(* Logix 5000 project; controller LeakTestAuto vendor 1 type 14 code 226 rev 37.11; software revision 37.01; part 8 of 12 *)
(* tags used below, declared in another part *)
   AOI_Conveyor_Seq : AOI_Sequencer_x64;
   AOI_CTS2 : AOI_CTS_INSTRUMENT;
   AOI_CTS2_Comms : AOI_CommStatus;
   AOI_CTS2_Seq : AOI_Sequencer_x64;
   AOI_Robot_Comms : AOI_CommStatus;
   AOI_RobotPos : AOI_RobotPositions;
   AOI_SeqSteps : AOI_StandardSeqSteps;
   Conveyor : udt_OutputStructure;
   Conveyor_Seq : udt_SequenceStructure_X64;
   ConveyorCleatSensorFault : BOOL;
   CTS2_BarcodeWrite : STRING80;
   CTS2_BasicResult : MESSAGE;
   CTS2_DataRead : STRING80;
   CTS2_DetailResult : MESSAGE;
   CTS2_Inputs : udt_CTS_INPUTS_FROM;
   CTS2_LastResultEval : STRING16;
   CTS2_LastTestUID : DINT;
   CTS2_NextTestUID : DINT;
   CTS2_NumTestsInSeq : SINT;
   CTS2_Outputs : udt_CTS_OUTPUTS_TO;
   CTS2_ReadMsg : MESSAGE;
   CTS2_Ready : DINT;
   CTS2_Result : udt_CTS_RESULT;
   CTS2_ResultHistoryLeak : udt_CTS_RESULT[10];
   CTS2_ResultHistoryVol : udt_CTS_RESULT[10];
   CTS2_Seq : udt_SequenceStructure_X64;
   CTS2_SeqUID : DINT;
   CTS2_UIDMsg : MESSAGE;
   CTS2_WriteMsg : MESSAGE;
   CTS_NoResult : udt_CTS_RESULT;
   CTS_ResultDump : udt_CTS_RESULT;
   CurrentDUTData : udt_DUTHistory[2];
   FFLU_CTS2Leak : CONTROL;
   FFLU_CTS2Vol : CONTROL;
   LeakTester2 : udt_OutputStructure;
   Mode_CapCTS : BOOL;
   Nest1Cylinder : udt_OutputStructure;
   Nest2Cylinder : udt_OutputStructure;
   ONS_CTS2ClearResultsBC : BOOL;
   ONS_CTS2GetResults : BOOL;
   ONS_CTS2ResultHistory : BOOL;
   ONS_RobotGripper : SINT;
   OP220 : udt_Mode;
   OP220_Seq : udt_SequenceStructure_X64;
   Robot : udt_OutputStructure;
   RobotGripper : udt_OutputStructure;
   RobotInputs : udt_EpsonInputs;
   RobotOutputs : udt_EpsonOutputs;
   TON_ConveyorCleatTimeout : TIMER;
   TON_ConvUnloadDelay : TIMER;
   TON_CTS2GetResultRetry : TIMER;
   TON_CTS2GetResultTimeout : TIMER;
   TON_CTS2NotGettingResultsTimeout : TIMER;
   TON_CTS2Trigger0 : TIMER;
   TON_CTS2Trigger1 : TIMER;
   TON_CTS2Trigger2 : TIMER;
   TON_Cylinder1DownTimeout : TIMER;
   TON_Cylinder1UpTimeout : TIMER;
   TON_Nest1CylinderTimer : TIMER;
   TON_RobotReqRetry : TIMER;
   TON_RobotReqTimeout : TIMER;
   ConveyorPurgeCounter : DINT;   // Outfeed Coveyor Purge Counter
   Delay_TMR : TIMER[11];   // Delay Timers
   I_OP220_N3_CONVEYOR_CLEAT : ALIAS FOR Local:3:I.Pt13.Data;
   I_OP220_N3_CONVEYOR_LOAD : ALIAS FOR Local:3:I.Pt12.Data;
   I_OP220_N3_CONVEYOR_UNLOAD : ALIAS FOR Local:3:I.Pt14.Data;
   I_OP220_N3_MAIN_AIR_OK : ALIAS FOR Local:3:I.Pt07.Data;
   I_OP220_N3_NEST1_EXTEND : ALIAS FOR Local:3:I.Pt04.Data;
   I_OP220_N3_NEST1_HOME : ALIAS FOR Local:3:I.Pt03.Data;
   I_OP220_N3_NEST2_HOME : ALIAS FOR Local:3:I.Pt05.Data;
   I_OP220_N3_REJECT_BIN_OK : ALIAS FOR Local:3:I.Pt09.Data;
   I_OP220_N4_CONVEYOR_ALARM_OK : ALIAS FOR Local:4:I.Pt03.Data;
   James_Dint : DINT;   // James Test Word
   O_OP220_N5_CONV_FWD : ALIAS FOR Local:5:O.Pt12.Data;
   O_OP220_N5_EN_CONV_ALM_RST : ALIAS FOR Local:5:O.Pt10.Data;
   O_OP220_N5_EN_GRIPPER_GRIP : ALIAS FOR Local:5:O.Pt14.Data;
   O_OP220_N5_EN_GRIPPER_UNGRIP : ALIAS FOR Local:5:O.Pt15.Data;
   O_OP220_N5_EN_NEST1_EXT : ALIAS FOR Local:5:O.Pt05.Data;
   O_OP220_N5_EN_NEST1_HOME : ALIAS FOR Local:5:O.Pt06.Data;
   Oneshot : DINT;   // Oneshots
   OP220_ConsumedFromMain_RobotPickupSafe : BOOL;
   PLC : AOI_PLC;
   ST1_Ignition_DataReady_Setup : BOOL;
   ST2_Ignition_DataReady_Setup : BOOL;
(* MainProgram, continued *)

ROUTINE R31_LeakTester2   (* ladder *)
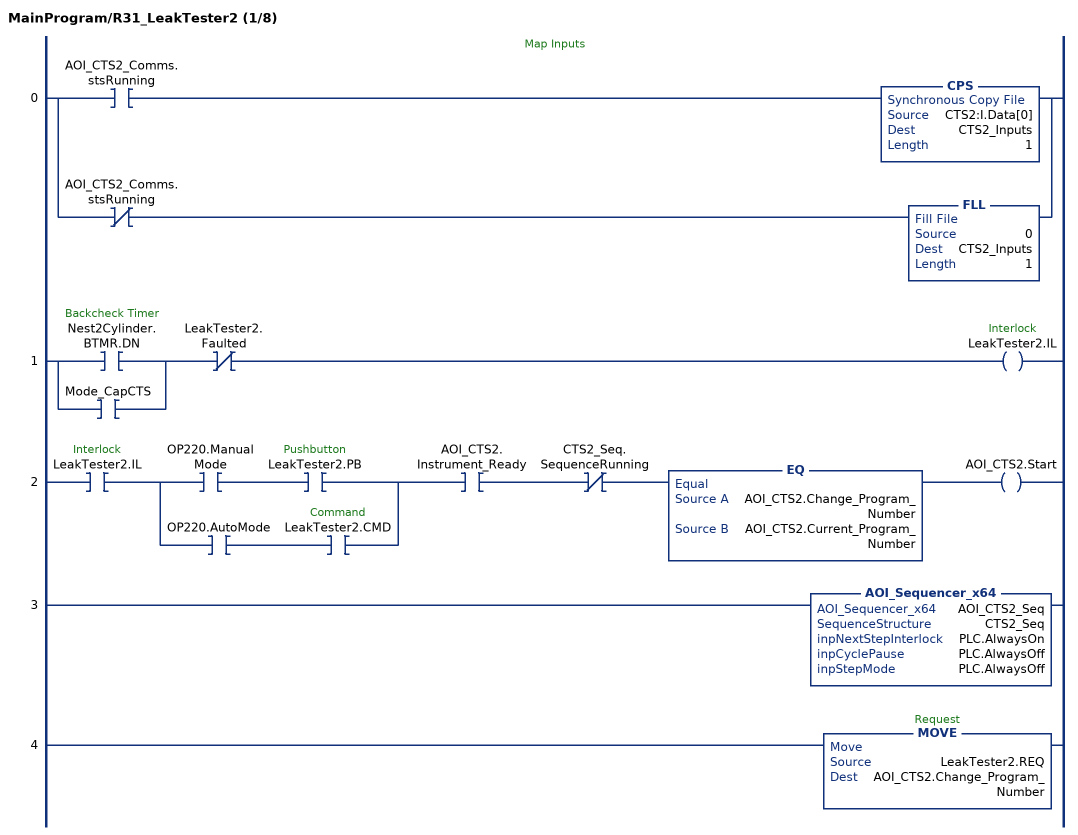
   // Map Inputs
   0: [XIC(AOI_CTS2_Comms.stsRunning) CPS(CTS2:I.Data[0],CTS2_Inputs,1) ,XIO(AOI_CTS2_Comms.stsRunning) FLL(0,CTS2_Inputs,1) ];
   1: [XIC(Nest2Cylinder.BTMR.DN) ,XIC(Mode_CapCTS) ]XIO(LeakTester2.Faulted)OTE(LeakTester2.IL);
   2: XIC(LeakTester2.IL)[XIC(OP220.ManualMode) XIC(LeakTester2.PB) ,XIC(OP220.AutoMode) XIC(LeakTester2.CMD) ]XIC(AOI_CTS2.Instrument_Ready)XIO(CTS2_Seq.SequenceRunning)EQ(AOI_CTS2.Change_Program_Number,AOI_CTS2.Current_Program_Number)OTE(AOI_CTS2.Start);
   3: AOI_Sequencer_x64(AOI_CTS2_Seq,CTS2_Seq,PLC.AlwaysOn,PLC.AlwaysOff,PLC.AlwaysOff);
   4: MOVE(LeakTester2.REQ,AOI_CTS2.Change_Program_Number);
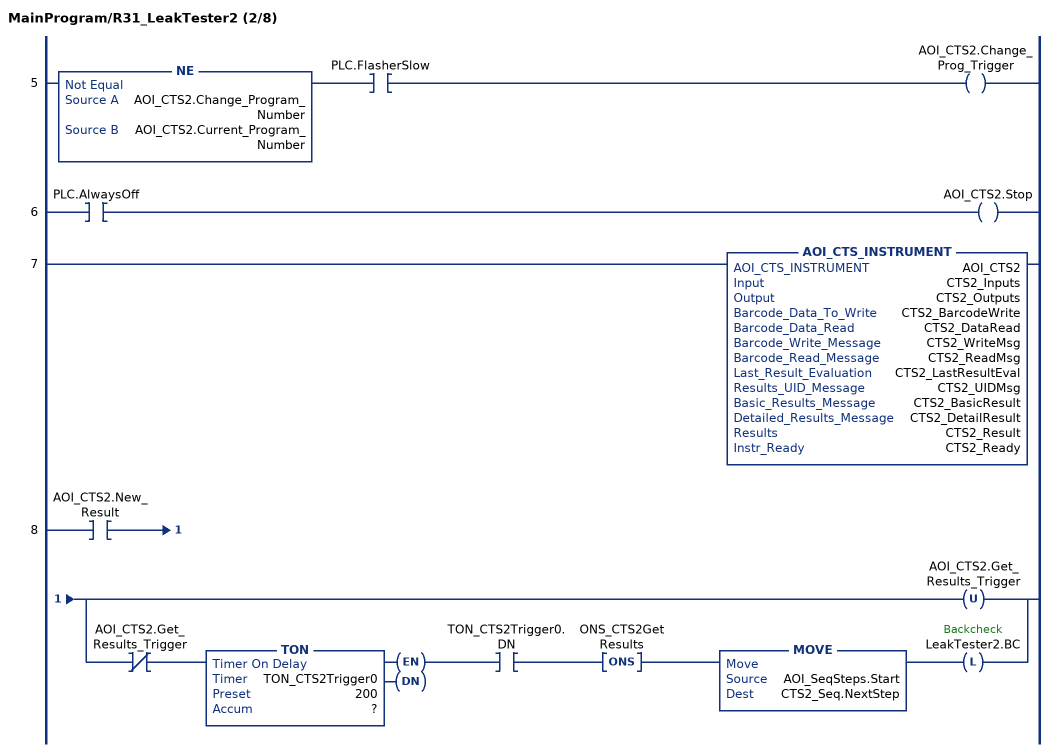
   5: NE(AOI_CTS2.Change_Program_Number,AOI_CTS2.Current_Program_Number)XIC(PLC.FlasherSlow)OTE(AOI_CTS2.Change_Prog_Trigger);
   6: XIC(PLC.AlwaysOff)OTE(AOI_CTS2.Stop);
   7: AOI_CTS_INSTRUMENT(AOI_CTS2,CTS2_Inputs,CTS2_Outputs,CTS2_BarcodeWrite,CTS2_DataRead,CTS2_WriteMsg,CTS2_ReadMsg,CTS2_LastResultEval,CTS2_UIDMsg,CTS2_BasicResult,CTS2_DetailResult,CTS2_Result,CTS2_Ready);
   8: XIC(AOI_CTS2.New_Result)[OTU(AOI_CTS2.Get_Results_Trigger) ,XIO(AOI_CTS2.Get_Results_Trigger) TON(TON_CTS2Trigger0,?,?) XIC(TON_CTS2Trigger0.DN) ONS(ONS_CTS2GetResults) MOVE(AOI_SeqSteps.Start,CTS2_Seq.NextStep) OTL(LeakTester2.BC) ];
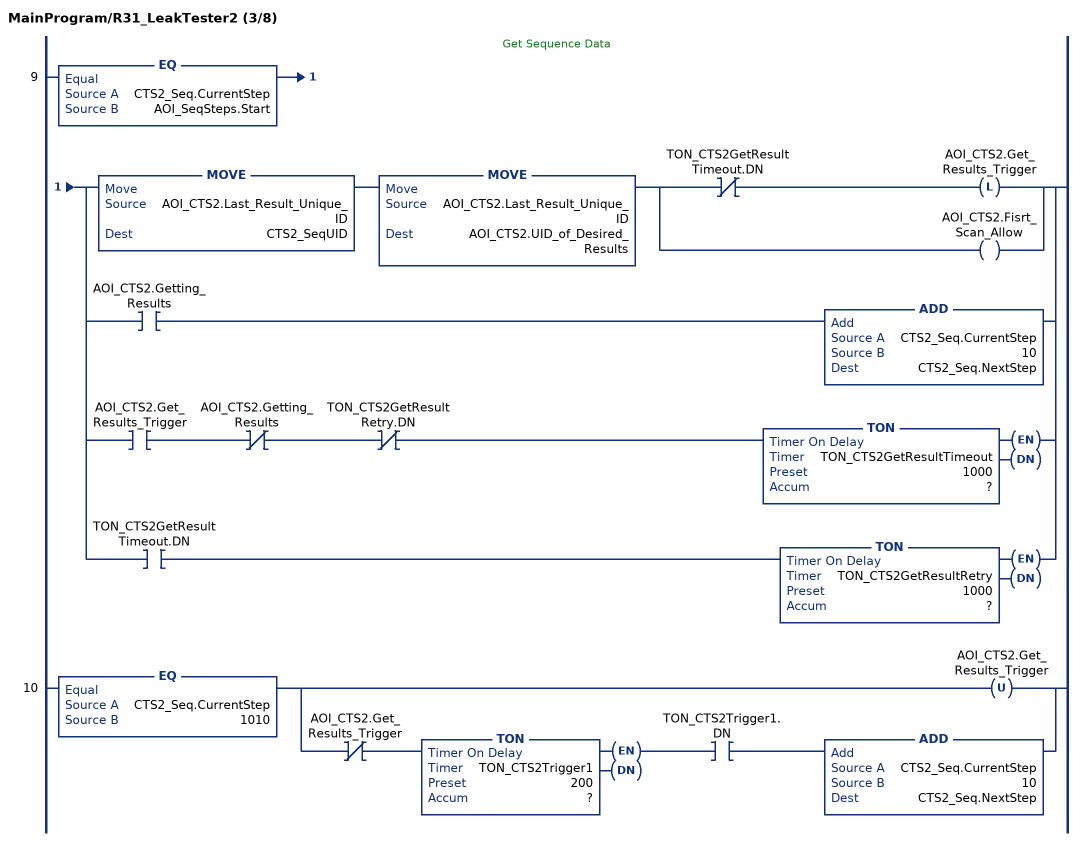
   // Get Sequence Data
   9: EQ(CTS2_Seq.CurrentStep,AOI_SeqSteps.Start)[MOVE(AOI_CTS2.Last_Result_Unique_ID,CTS2_SeqUID) MOVE(AOI_CTS2.Last_Result_Unique_ID,AOI_CTS2.UID_of_Desired_Results) [XIO(TON_CTS2GetResultTimeout.DN) OTL(AOI_CTS2.Get_Results_Trigger) ,OTE(AOI_CTS2.Fisrt_Scan_Allow) ] ,XIC(AOI_CTS2.Getting_Results) ADD(CTS2_Seq.CurrentStep,10,CTS2_Seq.NextStep) ,XIC(AOI_CTS2.Get_Results_Trigger) XIO(AOI_CTS2.Getting_Results) XIO(TON_CTS2GetResultRetry.DN) TON(TON_CTS2GetResultTimeout,?,?) ,XIC(TON_CTS2GetResultTimeout.DN) TON(TON_CTS2GetResultRetry,?,?) ];
   10: EQ(CTS2_Seq.CurrentStep,1010)[OTU(AOI_CTS2.Get_Results_Trigger) ,XIO(AOI_CTS2.Get_Results_Trigger) TON(TON_CTS2Trigger1,?,?) XIC(TON_CTS2Trigger1.DN) ADD(CTS2_Seq.CurrentStep,10,CTS2_Seq.NextStep) ];
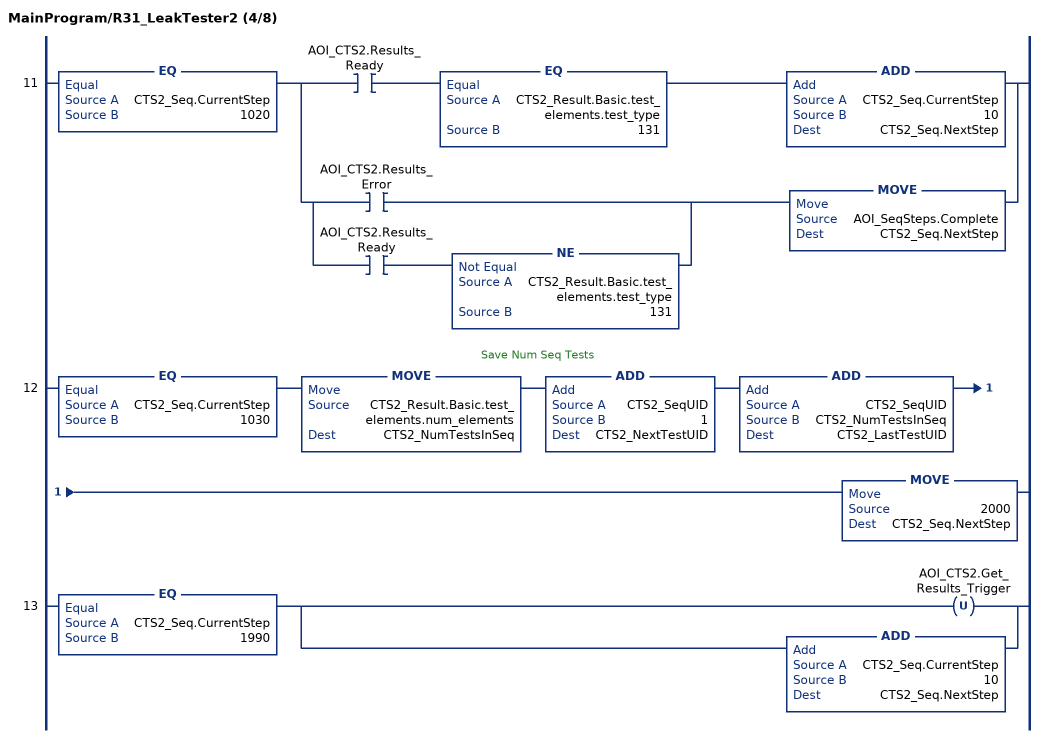
   11: EQ(CTS2_Seq.CurrentStep,1020)[XIC(AOI_CTS2.Results_Ready) EQ(CTS2_Result.Basic.test_elements.test_type,131) ADD(CTS2_Seq.CurrentStep,10,CTS2_Seq.NextStep) ,[XIC(AOI_CTS2.Results_Error) ,XIC(AOI_CTS2.Results_Ready) NE(CTS2_Result.Basic.test_elements.test_type,131) ] MOVE(AOI_SeqSteps.Complete,CTS2_Seq.NextStep) ];
   // Save Num Seq Tests
   12: EQ(CTS2_Seq.CurrentStep,1030)MOVE(CTS2_Result.Basic.test_elements.num_elements,CTS2_NumTestsInSeq)ADD(CTS2_SeqUID,1,CTS2_NextTestUID)ADD(CTS2_SeqUID,CTS2_NumTestsInSeq,CTS2_LastTestUID)MOVE(2000,CTS2_Seq.NextStep);
   13: EQ(CTS2_Seq.CurrentStep,1990)[OTU(AOI_CTS2.Get_Results_Trigger) ,ADD(CTS2_Seq.CurrentStep,10,CTS2_Seq.NextStep) ];
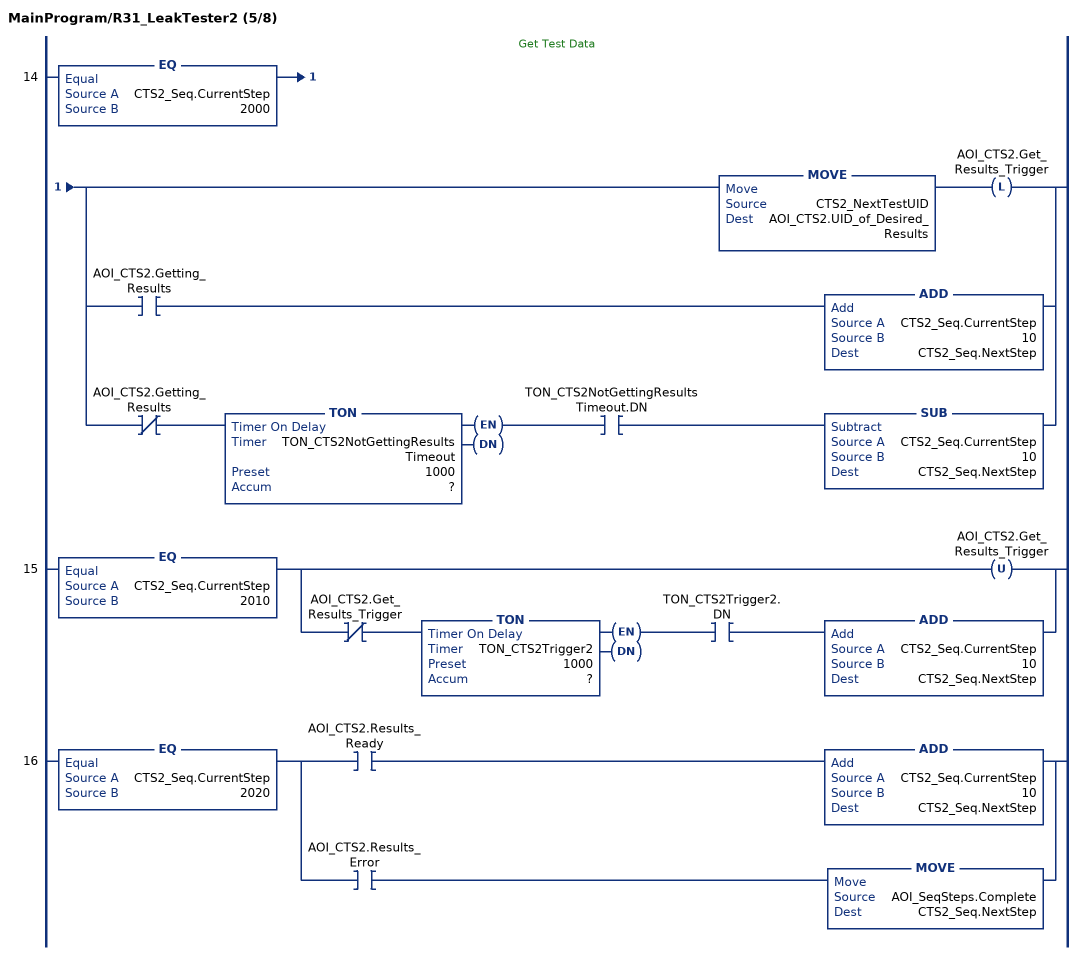
   // Get Test Data
   14: EQ(CTS2_Seq.CurrentStep,2000)[MOVE(CTS2_NextTestUID,AOI_CTS2.UID_of_Desired_Results) OTL(AOI_CTS2.Get_Results_Trigger) ,XIC(AOI_CTS2.Getting_Results) ADD(CTS2_Seq.CurrentStep,10,CTS2_Seq.NextStep) ,XIO(AOI_CTS2.Getting_Results) TON(TON_CTS2NotGettingResultsTimeout,?,?) XIC(TON_CTS2NotGettingResultsTimeout.DN) SUB(CTS2_Seq.CurrentStep,10,CTS2_Seq.NextStep) ];
   15: EQ(CTS2_Seq.CurrentStep,2010)[OTU(AOI_CTS2.Get_Results_Trigger) ,XIO(AOI_CTS2.Get_Results_Trigger) TON(TON_CTS2Trigger2,?,?) XIC(TON_CTS2Trigger2.DN) ADD(CTS2_Seq.CurrentStep,10,CTS2_Seq.NextStep) ];
   16: EQ(CTS2_Seq.CurrentStep,2020)[XIC(AOI_CTS2.Results_Ready) ADD(CTS2_Seq.CurrentStep,10,CTS2_Seq.NextStep) ,XIC(AOI_CTS2.Results_Error) MOVE(AOI_SeqSteps.Complete,CTS2_Seq.NextStep) ];
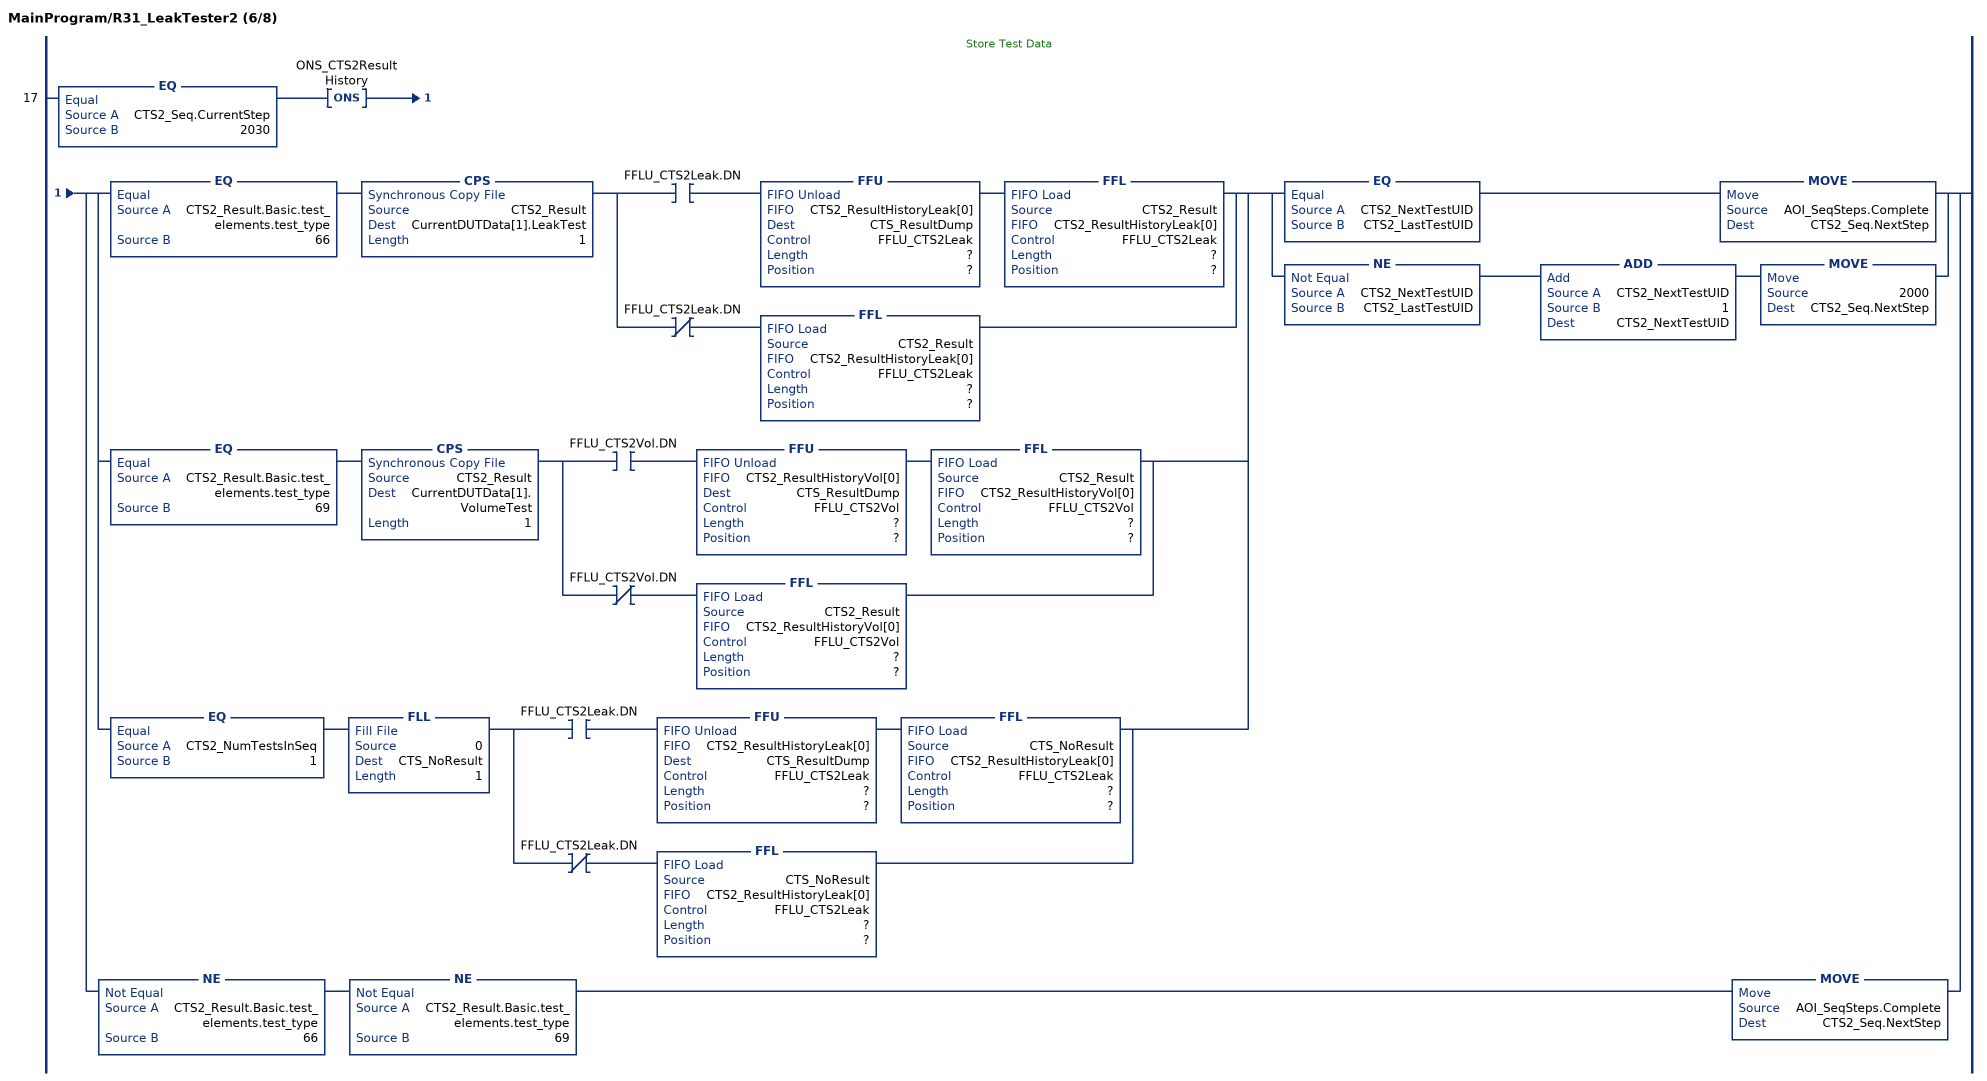
   // Store Test Data
   17: EQ(CTS2_Seq.CurrentStep,2030)ONS(ONS_CTS2ResultHistory)[[EQ(CTS2_Result.Basic.test_elements.test_type,66) CPS(CTS2_Result,CurrentDUTData[1].LeakTest,1) [XIC(FFLU_CTS2Leak.DN) FFU(CTS2_ResultHistoryLeak[0],CTS_ResultDump,FFLU_CTS2Leak,?,?) FFL(CTS2_Result,CTS2_ResultHistoryLeak[0],FFLU_CTS2Leak,?,?) ,XIO(FFLU_CTS2Leak.DN) FFL(CTS2_Result,CTS2_ResultHistoryLeak[0],FFLU_CTS2Leak,?,?) ] ,EQ(CTS2_Result.Basic.test_elements.test_type,69) CPS(CTS2_Result,CurrentDUTData[1].VolumeTest,1) [XIC(FFLU_CTS2Vol.DN) FFU(CTS2_ResultHistoryVol[0],CTS_ResultDump,FFLU_CTS2Vol,?,?) FFL(CTS2_Result,CTS2_ResultHistoryVol[0],FFLU_CTS2Vol,?,?) ,XIO(FFLU_CTS2Vol.DN) FFL(CTS2_Result,CTS2_ResultHistoryVol[0],FFLU_CTS2Vol,?,?) ] ,EQ(CTS2_NumTestsInSeq,1) FLL(0,CTS_NoResult,1) [XIC(FFLU_CTS2Leak.DN) FFU(CTS2_ResultHistoryLeak[0],CTS_ResultDump,FFLU_CTS2Leak,?,?) FFL(CTS_NoResult,CTS2_ResultHistoryLeak[0],FFLU_CTS2Leak,?,?) ,XIO(FFLU_CTS2Leak.DN) FFL(CTS_NoResult,CTS2_ResultHistoryLeak[0],FFLU_CTS2Leak,?,?) ] ] [EQ(CTS2_NextTestUID,CTS2_LastTestUID) MOVE(AOI_SeqSteps.Complete,CTS2_Seq.NextStep) ,NE(CTS2_NextTestUID,CTS2_LastTestUID) ADD(CTS2_NextTestUID,1,CTS2_NextTestUID) MOVE(2000,CTS2_Seq.NextStep) ] ,NE(CTS2_Result.Basic.test_elements.test_type,66) NE(CTS2_Result.Basic.test_elements.test_type,69) MOVE(AOI_SeqSteps.Complete,CTS2_Seq.NextStep) ];
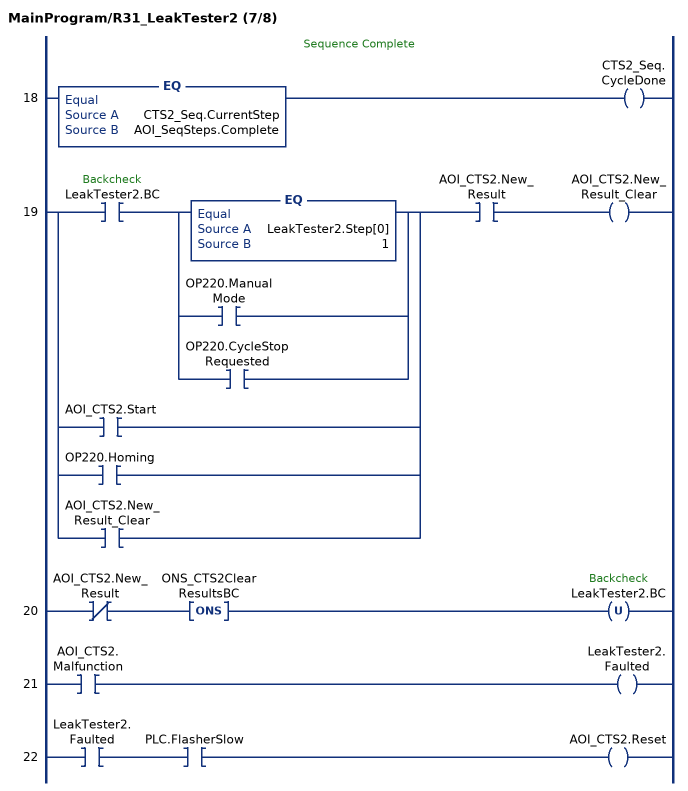
   // Sequence Complete
   18: EQ(CTS2_Seq.CurrentStep,AOI_SeqSteps.Complete)OTE(CTS2_Seq.CycleDone);
   19: [XIC(LeakTester2.BC) [EQ(LeakTester2.Step[0],1) ,XIC(OP220.ManualMode) ,XIC(OP220.CycleStopRequested) ] ,XIC(AOI_CTS2.Start) ,XIC(OP220.Homing) ,XIC(AOI_CTS2.New_Result_Clear) ]XIC(AOI_CTS2.New_Result)OTE(AOI_CTS2.New_Result_Clear);
   20: XIO(AOI_CTS2.New_Result)ONS(ONS_CTS2ClearResultsBC)OTU(LeakTester2.BC);
   21: XIC(AOI_CTS2.Malfunction)OTE(LeakTester2.Faulted);
   22: XIC(LeakTester2.Faulted)XIC(PLC.FlasherSlow)OTE(AOI_CTS2.Reset);
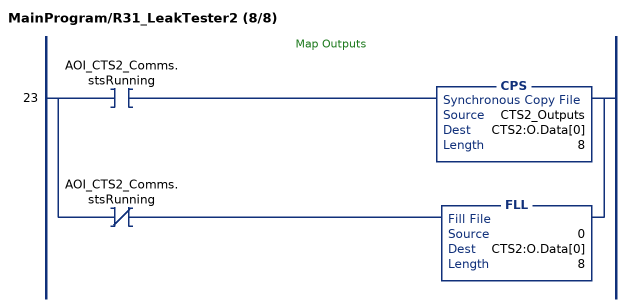
   // Map Outputs
   23: [XIC(AOI_CTS2_Comms.stsRunning) CPS(CTS2_Outputs,CTS2:O.Data[0],8) ,XIO(AOI_CTS2_Comms.stsRunning) FLL(0,CTS2:O.Data[0],8) ];
END_ROUTINE

ROUTINE R40_Robot   (* ladder *)
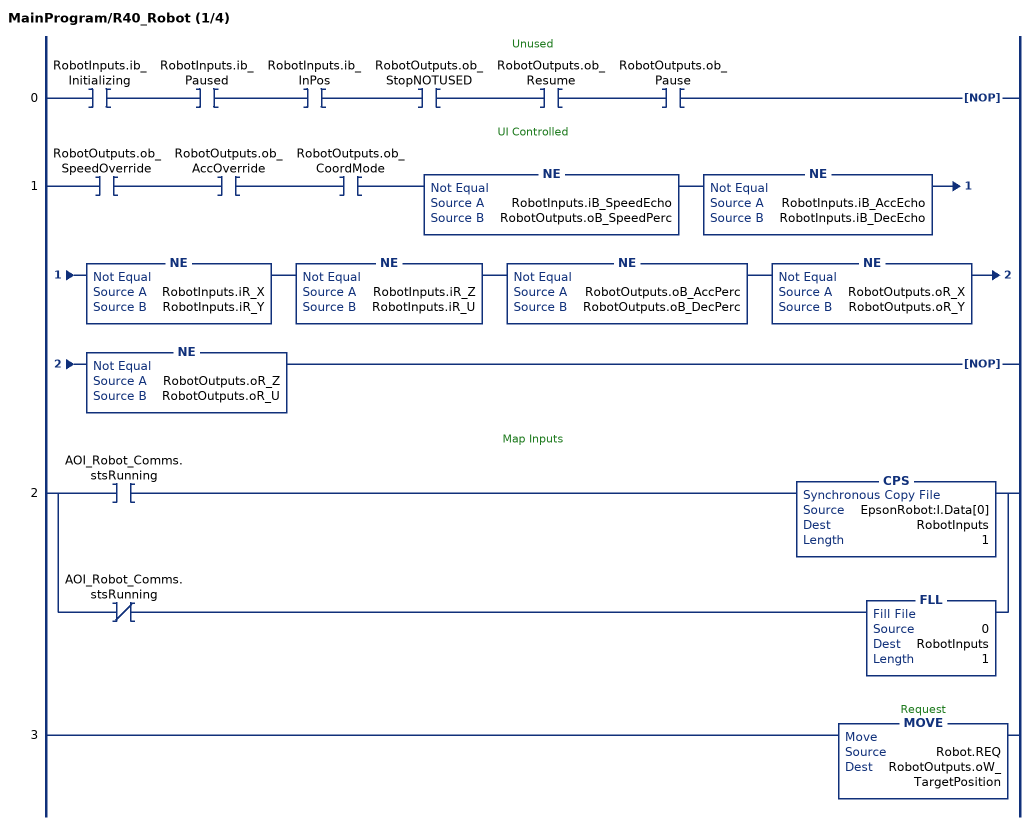
   // Unused
   0: XIC(RobotInputs.ib_Initializing)XIC(RobotInputs.ib_Paused)XIC(RobotInputs.ib_InPos)XIC(RobotOutputs.ob_StopNOTUSED)XIC(RobotOutputs.ob_Resume)XIC(RobotOutputs.ob_Pause)NOP();
   // UI Controlled
   1: XIC(RobotOutputs.ob_SpeedOverride)XIC(RobotOutputs.ob_AccOverride)XIC(RobotOutputs.ob_CoordMode)NE(RobotInputs.iB_SpeedEcho,RobotOutputs.oB_SpeedPerc)NE(RobotInputs.iB_AccEcho,RobotInputs.iB_DecEcho)NE(RobotInputs.iR_X,RobotInputs.iR_Y)NE(RobotInputs.iR_Z,RobotInputs.iR_U)NE(RobotOutputs.oB_AccPerc,RobotOutputs.oB_DecPerc)NE(RobotOutputs.oR_X,RobotOutputs.oR_Y)NE(RobotOutputs.oR_Z,RobotOutputs.oR_U)NOP();
   // Map Inputs
   2: [XIC(AOI_Robot_Comms.stsRunning) CPS(EpsonRobot:I.Data[0],RobotInputs,1) ,XIO(AOI_Robot_Comms.stsRunning) FLL(0,RobotInputs,1) ];
   3: MOVE(Robot.REQ,RobotOutputs.oW_TargetPosition);
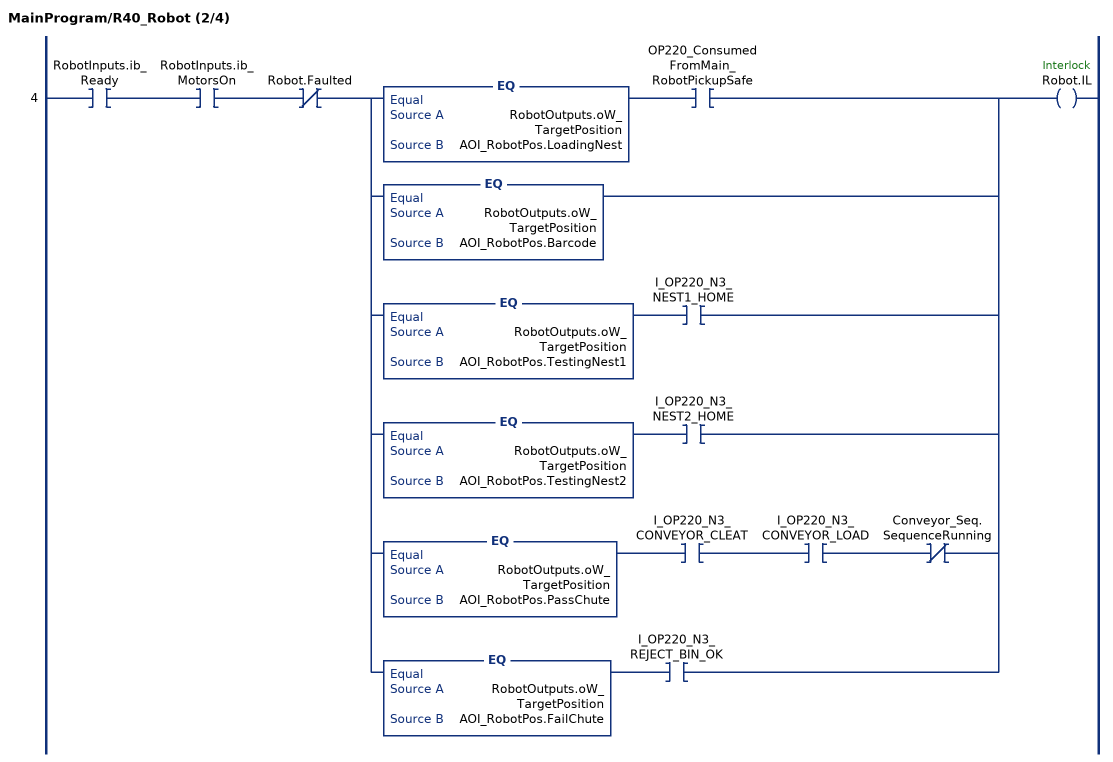
   4: XIC(RobotInputs.ib_Ready)XIC(RobotInputs.ib_MotorsOn)XIO(Robot.Faulted)[EQ(RobotOutputs.oW_TargetPosition,AOI_RobotPos.LoadingNest) XIC(OP220_ConsumedFromMain_RobotPickupSafe) ,EQ(RobotOutputs.oW_TargetPosition,AOI_RobotPos.Barcode) ,EQ(RobotOutputs.oW_TargetPosition,AOI_RobotPos.TestingNest1) XIC(I_OP220_N3_NEST1_HOME) ,EQ(RobotOutputs.oW_TargetPosition,AOI_RobotPos.TestingNest2) XIC(I_OP220_N3_NEST2_HOME) ,EQ(RobotOutputs.oW_TargetPosition,AOI_RobotPos.PassChute) XIC(I_OP220_N3_CONVEYOR_CLEAT) XIC(I_OP220_N3_CONVEYOR_LOAD) XIO(Conveyor_Seq.SequenceRunning) ,EQ(RobotOutputs.oW_TargetPosition,AOI_RobotPos.FailChute) XIC(I_OP220_N3_REJECT_BIN_OK) ]OTE(Robot.IL);
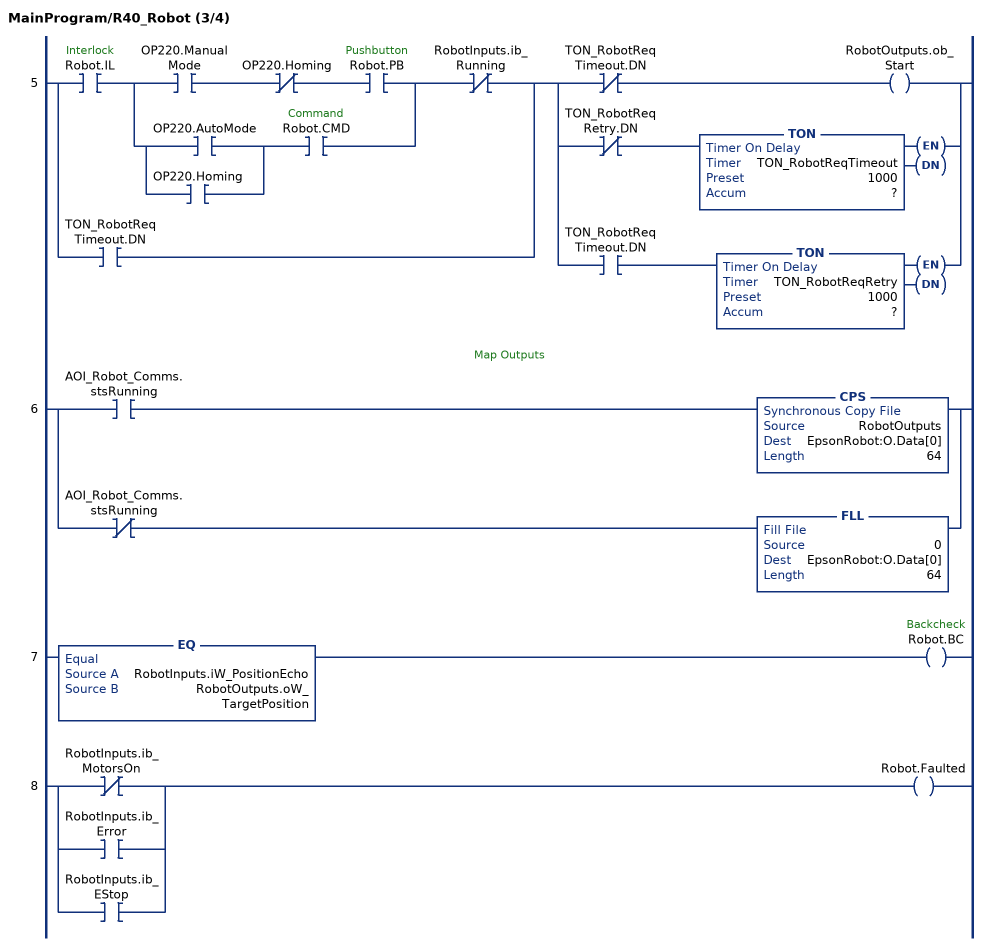
   5: [XIC(Robot.IL) [XIC(OP220.ManualMode) XIO(OP220.Homing) XIC(Robot.PB) ,[XIC(OP220.AutoMode) ,XIC(OP220.Homing) ] XIC(Robot.CMD) ] XIO(RobotInputs.ib_Running) ,XIC(TON_RobotReqTimeout.DN) ][XIO(TON_RobotReqTimeout.DN) OTE(RobotOutputs.ob_Start) ,XIO(TON_RobotReqRetry.DN) TON(TON_RobotReqTimeout,?,?) ,XIC(TON_RobotReqTimeout.DN) TON(TON_RobotReqRetry,?,?) ];
   // Map Outputs
   6: [XIC(AOI_Robot_Comms.stsRunning) CPS(RobotOutputs,EpsonRobot:O.Data[0],64) ,XIO(AOI_Robot_Comms.stsRunning) FLL(0,EpsonRobot:O.Data[0],64) ];
   7: EQ(RobotInputs.iW_PositionEcho,RobotOutputs.oW_TargetPosition)OTE(Robot.BC);
   8: [XIO(RobotInputs.ib_MotorsOn) ,XIC(RobotInputs.ib_Error) ,XIC(RobotInputs.ib_EStop) ]OTE(Robot.Faulted);
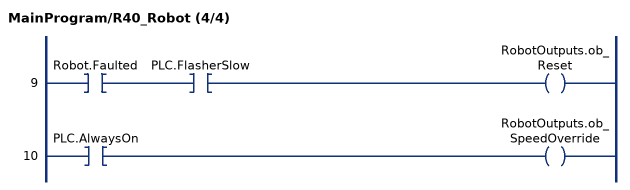
   9: XIC(Robot.Faulted)XIC(PLC.FlasherSlow)OTE(RobotOutputs.ob_Reset);
   10: XIC(PLC.AlwaysOn)OTE(RobotOutputs.ob_SpeedOverride);
END_ROUTINE

ROUTINE R41_RobotGripper   (* ladder *)
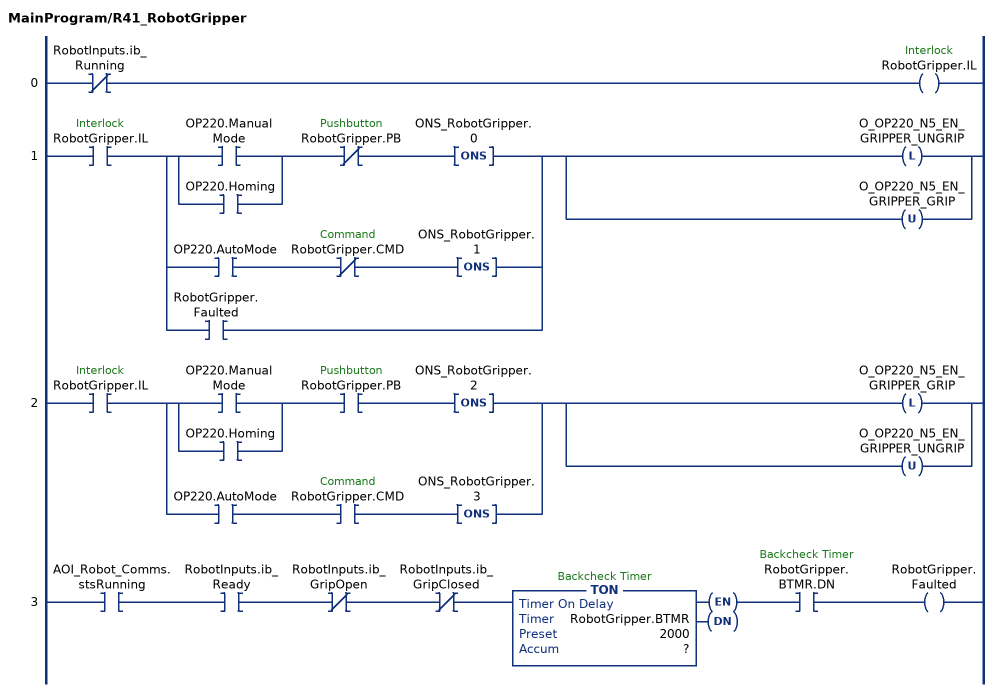
   0: XIO(RobotInputs.ib_Running)OTE(RobotGripper.IL);
   1: XIC(RobotGripper.IL)[[[XIC(OP220.ManualMode) ,XIC(OP220.Homing) ] XIO(RobotGripper.PB) ONS(ONS_RobotGripper.0) ,XIC(OP220.AutoMode) XIO(RobotGripper.CMD) ONS(ONS_RobotGripper.1) ] ,XIC(RobotGripper.Faulted) ][OTL(O_OP220_N5_EN_GRIPPER_UNGRIP) ,OTU(O_OP220_N5_EN_GRIPPER_GRIP) ];
   2: XIC(RobotGripper.IL)[[XIC(OP220.ManualMode) ,XIC(OP220.Homing) ] XIC(RobotGripper.PB) ONS(ONS_RobotGripper.2) ,XIC(OP220.AutoMode) XIC(RobotGripper.CMD) ONS(ONS_RobotGripper.3) ][OTL(O_OP220_N5_EN_GRIPPER_GRIP) ,OTU(O_OP220_N5_EN_GRIPPER_UNGRIP) ];
   3: XIC(AOI_Robot_Comms.stsRunning)XIC(RobotInputs.ib_Ready)XIO(RobotInputs.ib_GripOpen)XIO(RobotInputs.ib_GripClosed)TON(RobotGripper.BTMR,?,?)XIC(RobotGripper.BTMR.DN)OTE(RobotGripper.Faulted);
END_ROUTINE

ROUTINE R50_Conveyor   (* ladder *)
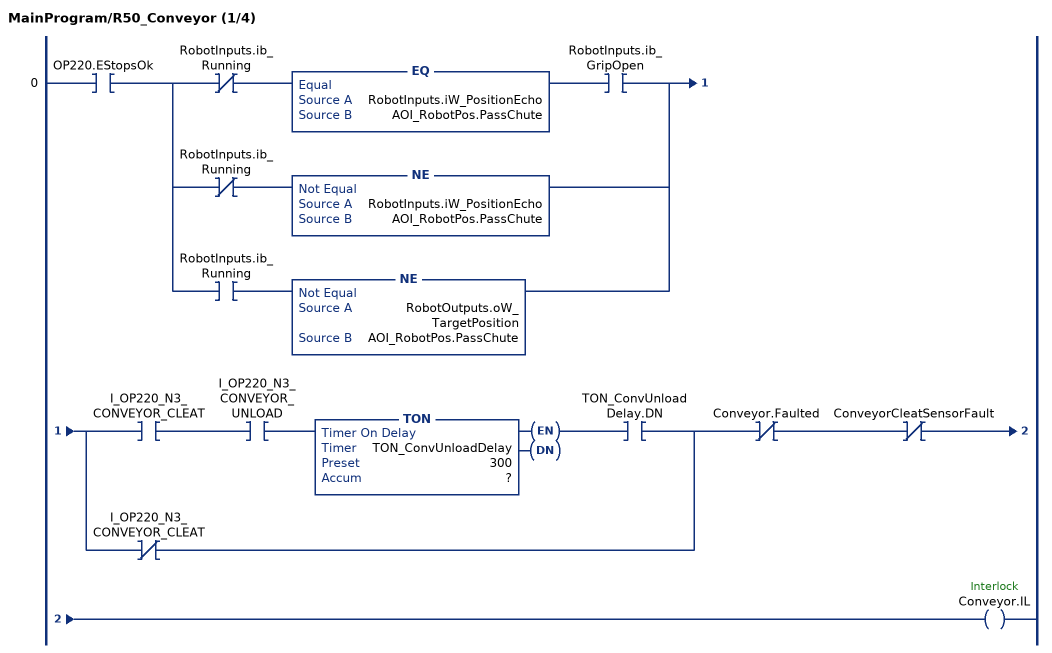
   0: XIC(OP220.EStopsOk)[XIO(RobotInputs.ib_Running) EQ(RobotInputs.iW_PositionEcho,AOI_RobotPos.PassChute) XIC(RobotInputs.ib_GripOpen) ,XIO(RobotInputs.ib_Running) NE(RobotInputs.iW_PositionEcho,AOI_RobotPos.PassChute) ,XIC(RobotInputs.ib_Running) NE(RobotOutputs.oW_TargetPosition,AOI_RobotPos.PassChute) ][XIC(I_OP220_N3_CONVEYOR_CLEAT) XIC(I_OP220_N3_CONVEYOR_UNLOAD) TON(TON_ConvUnloadDelay,?,?) XIC(TON_ConvUnloadDelay.DN) ,XIO(I_OP220_N3_CONVEYOR_CLEAT) ]XIO(Conveyor.Faulted)XIO(ConveyorCleatSensorFault)OTE(Conveyor.IL);
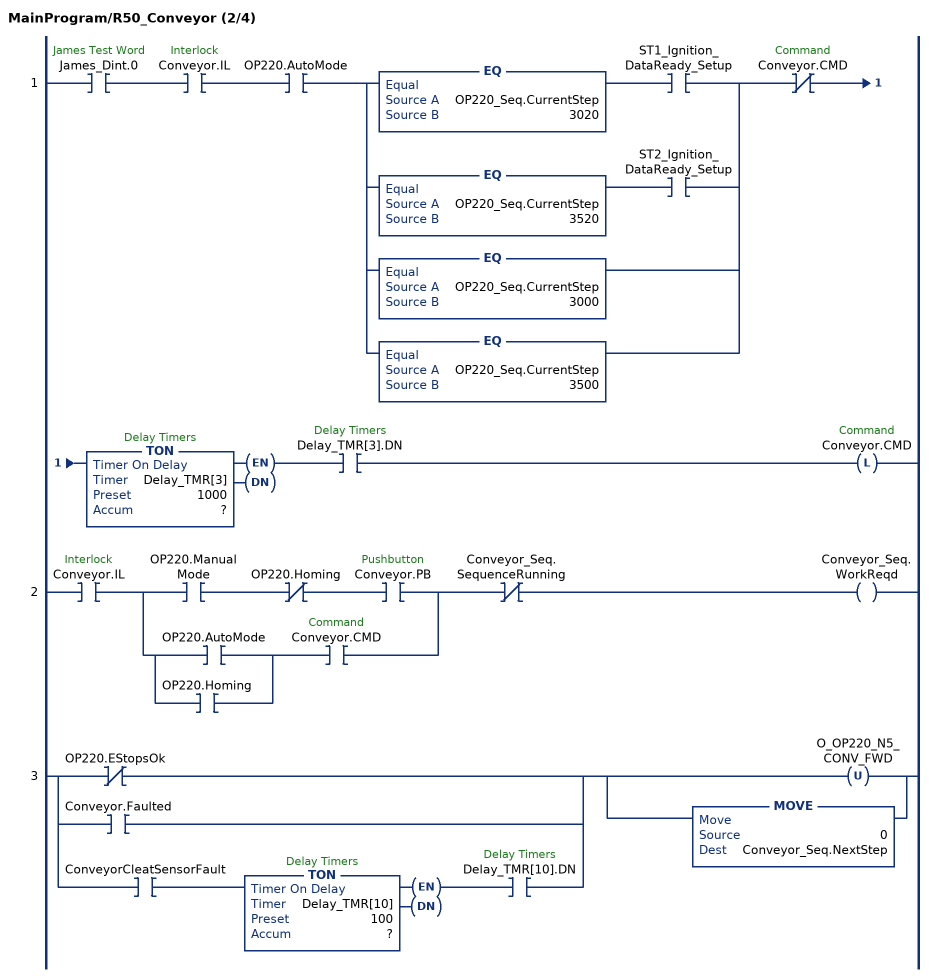
   1: XIC(James_Dint.0)XIC(Conveyor.IL)XIC(OP220.AutoMode)[EQ(OP220_Seq.CurrentStep,3020) XIC(ST1_Ignition_DataReady_Setup) ,EQ(OP220_Seq.CurrentStep,3520) XIC(ST2_Ignition_DataReady_Setup) ,EQ(OP220_Seq.CurrentStep,3000) ,EQ(OP220_Seq.CurrentStep,3500) ]XIO(Conveyor.CMD)TON(Delay_TMR[3],?,?)XIC(Delay_TMR[3].DN)OTL(Conveyor.CMD);
   2: XIC(Conveyor.IL)[XIC(OP220.ManualMode) XIO(OP220.Homing) XIC(Conveyor.PB) ,[XIC(OP220.AutoMode) ,XIC(OP220.Homing) ] XIC(Conveyor.CMD) ]XIO(Conveyor_Seq.SequenceRunning)OTE(Conveyor_Seq.WorkReqd);
   3: [XIO(OP220.EStopsOk) ,XIC(Conveyor.Faulted) ,XIC(ConveyorCleatSensorFault) TON(Delay_TMR[10],?,?) XIC(Delay_TMR[10].DN) ][OTU(O_OP220_N5_CONV_FWD) ,MOVE(0,Conveyor_Seq.NextStep) ];
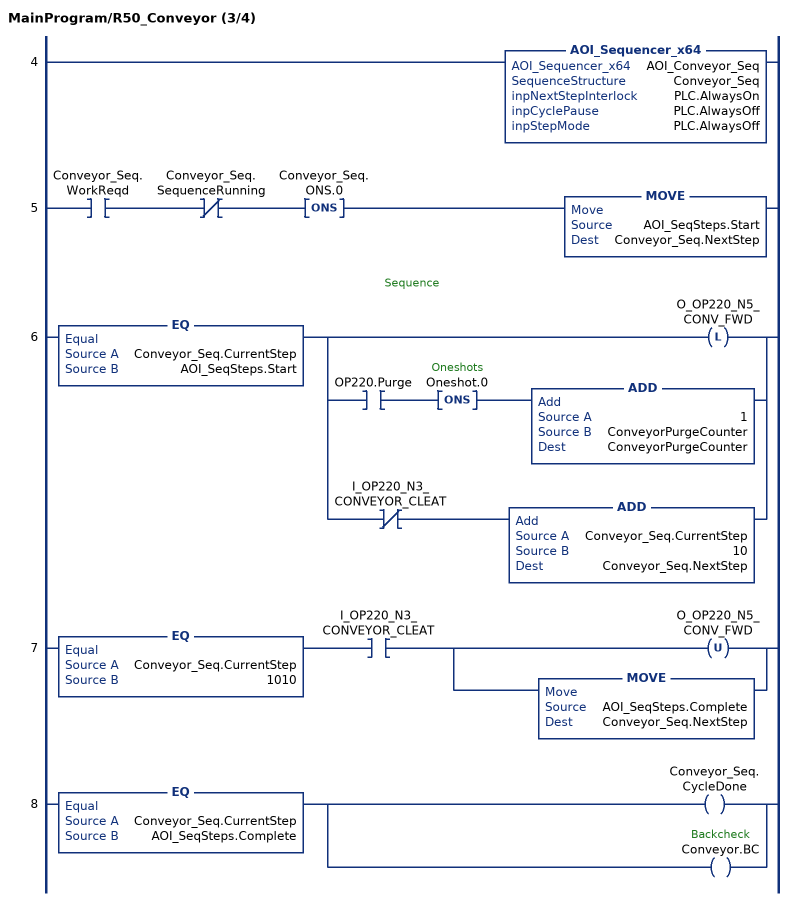
   4: AOI_Sequencer_x64(AOI_Conveyor_Seq,Conveyor_Seq,PLC.AlwaysOn,PLC.AlwaysOff,PLC.AlwaysOff);
   5: XIC(Conveyor_Seq.WorkReqd)XIO(Conveyor_Seq.SequenceRunning)ONS(Conveyor_Seq.ONS.0)MOVE(AOI_SeqSteps.Start,Conveyor_Seq.NextStep);
   // Sequence
   6: EQ(Conveyor_Seq.CurrentStep,AOI_SeqSteps.Start)[OTL(O_OP220_N5_CONV_FWD) ,XIC(OP220.Purge) ONS(Oneshot.0) ADD(1,ConveyorPurgeCounter,ConveyorPurgeCounter) ,XIO(I_OP220_N3_CONVEYOR_CLEAT) ADD(Conveyor_Seq.CurrentStep,10,Conveyor_Seq.NextStep) ];
   7: EQ(Conveyor_Seq.CurrentStep,1010)XIC(I_OP220_N3_CONVEYOR_CLEAT)[OTU(O_OP220_N5_CONV_FWD) ,MOVE(AOI_SeqSteps.Complete,Conveyor_Seq.NextStep) ];
   8: EQ(Conveyor_Seq.CurrentStep,AOI_SeqSteps.Complete)[OTE(Conveyor_Seq.CycleDone) ,OTE(Conveyor.BC) ];
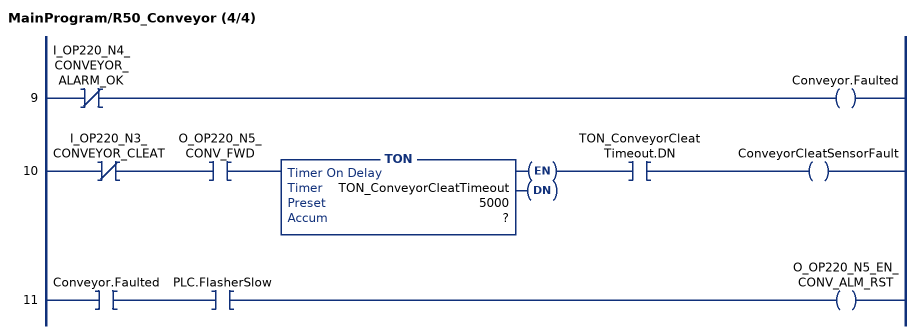
   9: XIO(I_OP220_N4_CONVEYOR_ALARM_OK)OTE(Conveyor.Faulted);
   10: XIO(I_OP220_N3_CONVEYOR_CLEAT)XIC(O_OP220_N5_CONV_FWD)TON(TON_ConveyorCleatTimeout,?,?)XIC(TON_ConveyorCleatTimeout.DN)OTE(ConveyorCleatSensorFault);
   11: XIC(Conveyor.Faulted)XIC(PLC.FlasherSlow)OTE(O_OP220_N5_EN_CONV_ALM_RST);
END_ROUTINE

ROUTINE R60_Nest1Cylinder   (* ladder *)
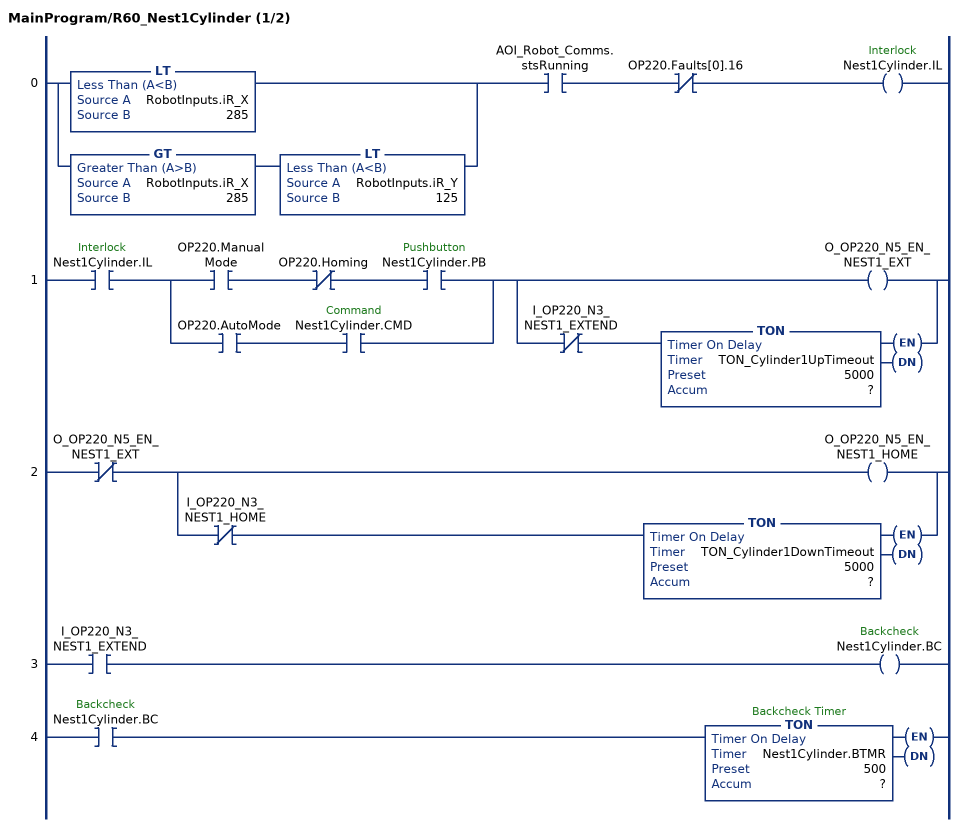
   0: [LT(RobotInputs.iR_X,285) ,GT(RobotInputs.iR_X,285) LT(RobotInputs.iR_Y,125) ]XIC(AOI_Robot_Comms.stsRunning)XIO(OP220.Faults[0].16)OTE(Nest1Cylinder.IL);
   1: XIC(Nest1Cylinder.IL)[XIC(OP220.ManualMode) XIO(OP220.Homing) XIC(Nest1Cylinder.PB) ,XIC(OP220.AutoMode) XIC(Nest1Cylinder.CMD) ][OTE(O_OP220_N5_EN_NEST1_EXT) ,XIO(I_OP220_N3_NEST1_EXTEND) TON(TON_Cylinder1UpTimeout,?,?) ];
   2: XIO(O_OP220_N5_EN_NEST1_EXT)[OTE(O_OP220_N5_EN_NEST1_HOME) ,XIO(I_OP220_N3_NEST1_HOME) TON(TON_Cylinder1DownTimeout,?,?) ];
   3: XIC(I_OP220_N3_NEST1_EXTEND)OTE(Nest1Cylinder.BC);
   4: XIC(Nest1Cylinder.BC)TON(Nest1Cylinder.BTMR,?,?);
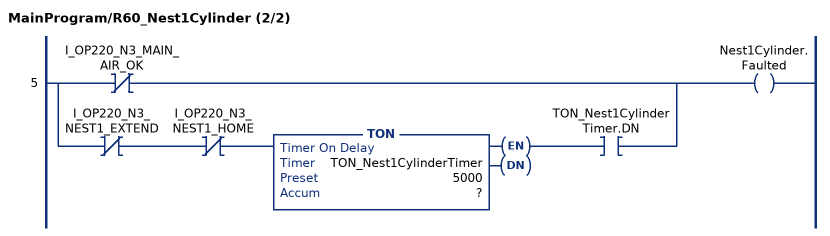
   5: [XIO(I_OP220_N3_MAIN_AIR_OK) ,XIO(I_OP220_N3_NEST1_EXTEND) XIO(I_OP220_N3_NEST1_HOME) TON(TON_Nest1CylinderTimer,?,?) XIC(TON_Nest1CylinderTimer.DN) ]OTE(Nest1Cylinder.Faulted);
END_ROUTINE
